// TIA Portal V18 export
TYPE "UDT_DLsDI"
// stored: IsFailsafeCompliant false
   STRUCT
      xDieselLineHeatingReady : Array[1..2] of Bool;
      xDieselLineHeatingInd : Array[1..2] of Bool;
      xDieselLinePumpInd : Array[1..2] of Bool;
      xDieselLinePnom : Bool;   // 10.67 Номінальний тиск в ДП ліній
      xDieselLineValveToBoilerInd : Bool;   // 10.66 Клапанна група на Котел
      xDieselLinePmax : Bool;   // 10.68 Високий тиск в ДП ліній
      xDieselLinePumpZoneWaterFloodAlarm : Bool;   // 10.79 Затоплення приямку з насосами
      xDieselLineMainTankDoubleWallAlarmInd : Bool;   // 10.63 62 SGB DL-4000
      xDieselLineMainTankMinLevelInd : Bool;   // 10.75 76
      Reserve1 : Bool;
      Reserve2 : Bool;
      xDieselLinePumpPanelSelectorOff : Bool;
      xDieselLinePumpPanelSelectorP1Man : Bool;
      xDieselLinePumpPanelSelectorP2Man : Bool;
      xDieselLinePumpPanelSelectorAuto : Bool;
   END_STRUCT;
END_TYPE
